FUNCTION_BLOCK ST_blinker
VAR_INPUT
	execute:BOOL;
	period: TIME := T#1S;
END_VAR
VAR_OUTPUT
	output:BOOL;
END_VAR
VAR
	delay: TON;
END_VAR

delay(IN := NOT delay.Q, PT := period / 2);
output := (NOT output AND delay.Q) OR (output AND NOT delay.Q) AND execute;

END_FUNCTION_BLOCK

(* stored: Version 1.1.0.1, ProductVersion 3.1.4024.12
   POU ST_blinker: Id {37e71a61-3e5c-44ed-a5e7-5d62c766e7fe}, SpecialFunc None *)
